(*
SPDX-FileCopyrightText: © 2026 Oleksandr Tiutyk <trofimich@gmail.com>
SPDX-License-Identifier: MIT
License: https://opensource.org/license/mit
*)

(*!
<summary>Reports an argument whose named type is not supported by the operation.</summary>
<description>
The caller detects the invalid argument. Throw records a diagnostic message and source metadata; it does not
inspect the actual argument or decide which types are supported. Dynamic instances belong to the current task
memory manager until cleanup. Dynamic copies are explicitly registered by Clone after construction; plain
__NEW does not transfer ownership to the task manager.
</description>
*)

{attribute 'enable_dynamic_creation'}
{attribute 'no_explicit_call' := 'do not call this function block directly'}
FUNCTION_BLOCK ArgumentTypeNotSupportedException EXTENDS GeneralException IMPLEMENTS IArgumentTypeNotSupportedException
VAR_STAT
	//! <summary>Class name shared by all instances of this function block.</summary>
	{attribute 'hide'} 
	_ClassName : STRING := __POUNAME();
END_VAR

{attribute 'monitoring' := 'call'}
PROPERTY ClassName : REFERENCE TO STRING
GET
ClassName REF= _ClassName;
END_GET
END_PROPERTY

(*!
<summary>Creates a distinct auto-disposed copy of this concrete exception type.</summary>
<description>
Copies message, code, source and timestamps through CopyGeneralFields; any prepared inner cause remains
borrowed. The current task memory manager owns the clone until cleanup. Allocation failure is terminal.
Descendants with additional payload must override Clone to preserve their type and fields. Registers the newly
constructed instance before copying payload, outside FB_init. Registration failure releases the unregistered
instance and raises a terminal error; copy failure leaves the registered instance owned by the task manager
for cleanup. Custom overrides must follow the same ownership sequence.
</description>
*)
METHOD Clone : IObject
VAR
	exceptionClone : POINTER TO ArgumentTypeNotSupportedException;
END_VAR
exceptionClone := __NEW(ArgumentTypeNotSupportedException);

IF exceptionClone = 0 THEN
	DynamicMemoryManager.RaiseAllocationFailure();
END_IF

DynamicMemoryManager.RegisterAutoDisposedObject(autoDisposedObject := exceptionClone^);

exceptionClone^.CopyGeneralFields(sourceException := THIS^);

Clone := exceptionClone^;
END_METHOD

(*!
<summary>Provides the library namespace used in diagnostics.</summary>
<description>
Borrowed read-only reference to the compiler-initialized library namespace; no ownership transfer.
</description>
*)
{attribute 'monitoring' := 'call'}
PROPERTY NamespaceName : REFERENCE TO STRING
GET
NamespaceName REF= CurrentNamespace.Name;
END_GET
END_PROPERTY

(*!
<summary>Reports the byte size of this concrete instance.</summary>
<description>
Uses XSIZEOF on the instance. Does not include separately allocated payloads or prove that an arbitrary
address is valid.
</description>
*)
{attribute 'monitoring' := 'call'}
PROPERTY SelfSize : ULINT
GET
SelfSize := XSIZEOF(THIS^);
END_GET
END_PROPERTY

(*!
<summary>Builds the argument diagnostic and propagates this exception.</summary>
<description>
Call in the owning cyclic task, not during FB_init. Captures message, source and timestamps with zero error
code and no inner cause. Supplied names are copied into a local buffer without heap allocation; no caller
storage is retained. Exception clone allocation failure follows the shared terminal memory mechanism.
</description>
<param name="argumentName">Name of the argument rejected by the caller.</param>
*)
METHOD Throw
VAR_INPUT
	sourceNamespaceName : STRING;
	sourceClassName : STRING;
	sourcePOUName : STRING;
	sourcePosition : STRING;
	argumentName : STRING;
	argumentTypeName : STRING;
END_VAR
VAR
	message : ERROR_MESSAGE;
END_VAR
WideStrings.Append255(
	message,
	"Argument '",
	TO_WSTRING(argumentName),
	"' has not supported type '",
	TO_WSTRING(argumentTypeName),
	"' in '",
	TO_WSTRING(GetFullPOUName(
		sourceNamespaceName := sourceNamespaceName,
		sourceClassName := sourceClassName,
		sourcePOUName := sourcePOUName
	)),
	"'");

InternalThrow(
	sourceNamespaceName := sourceNamespaceName,
	sourceClassName := sourceClassName,
	sourcePOUName := sourcePOUName,
	sourcePosition := sourcePosition,
	message := message,
	errorCode := 0,
	innerException := 0
);
END_METHOD

END_FUNCTION_BLOCK

(* stored: Version 1.1.0.1
   POU ArgumentTypeNotSupportedException: Id {e65e380b-db18-442f-96f6-e7cc3cbe0ecf}, SpecialFunc None
   Property ClassName: Id {c383e4ab-f205-4088-beec-3b49964add95}
   Get Get: Id {fbcface4-d006-407b-8285-9e6e1a6c721b}
   Method Clone: Id {fd83cf8f-f225-4457-8d29-4778b5e86181}
   Property NamespaceName: Id {c2f8462c-4e2b-4478-a643-70dd04cb396e}
   Get Get: Id {7a49ea9d-6355-4d21-9b38-2110e63f7f06}
   Property SelfSize: Id {69476834-9b65-418a-8c27-e88ba387485b}
   Get Get: Id {1d5c2309-da50-4022-bf9b-42e1a3854f65}
   Method Throw: Id {e14b9f6f-e370-4201-a21c-0513badf6b37} *)
